Staubli VAL3: FILEDIR.pjx

--- FILEDIR.pjx ---
Parameters version=s7.7.1 stackSize=5000 millimeterUnit=true
Program file=CloseAllFile.pgx
Program file=CloseFile.pgx
Program file=CopyFileContext.pgx
Program file=CreatDir.pgx
Program file=CreatFile.pgx
Program file=Example.pgx
Program file=ExampleTest.pgx
Program file=GetLine.pgx
Program file=GetTrajFlag.pgx
Program file=ReadMe.pgx
Program file=SplitActionLine.pgx
Program file=SplitCutPreset.pgx
Program file=SplitJoint.pgx
Program file=SplitMoveC.pgx
Program file=SplitMoveJ.pgx
Program file=SplitMoveL.pgx
Program file=SplitNumS.pgx
Program file=SplitPresetLine.pgx
Program file=SplitString.pgx
Program file=SplitTrsf.pgx
Program file=start.pgx
Program file=stop.pgx
Program file=WriteLine.pgx
Data file=FileDir.dtx

--- FILEDIR.dtx ---
mdesc mNomSpeed
num nFile2ID
num nFileID
string sBuff

--- start.pgx ---
program start()
begin
  call ExampleTest()
end

--- CloseAllFile.pgx ---
public program CloseAllFile()
begin

  call CloseFile(0)
  call CloseFile(1)
  call CloseFile(2)
  call CloseFile(3)
  call CloseFile(4)
  call CloseFile(5)
  call CloseFile(6)
  call CloseFile(7)
  call CloseFile(8)
  call CloseFile(9)
  delay(0)

end

--- CloseFile.pgx ---
public program CloseFile(num x_nFileID (dimensions=1))
begin

  //文件标志符


  if x_nFileID<0 or x_nFileID>9
    return
  endIf

  //
  switch x_nFileID
    case 0
      $fileClose(0)
    break

    case 1
      $fileClose(1)
    break

    case 2
      $fileClose(2)
    break

    case 3
      $fileClose(3)
    break

    case 4
      $fileClose(4)
    break

    case 5
      $fileClose(5)
    break
    case 6
      $fileClose(6)
    break

    case 7
      $fileClose(7)
    break
    case 8
      $fileClose(8)
    break

    case 9
      $fileClose(9)
    break


  endSwitch


end

--- CopyFileContext.pgx ---
public program CopyFileContext(bool x_bRes (dimensions=1), string x_sFileSource (dimensions=1), string x_sFileDest (dimensions=1), num x_nStart (dimensions=1), num x_nEnd (dimensions=1))
  local num l_nIndex
  local num l_nNum
  local string l_sBuff
begin

  x_bRes=false
  if x_nEnd==-1
    x_nEnd=50000000
  endIf
  if x_sFileDest=="" or x_nStart<0 or x_nEnd<1 or x_nEnd<x_nStart or x_sFileDest==""
    return
  endIf
  if !$fileExists(x_sFileSource) or !$fileExists(x_sFileDest)
    return
  endIf


  nFileID=$fileOpen(x_sFileSource,"r")
  if nFileID<0 or nFileID>9
    return
  endIf

  nFile2ID=$fileOpen(x_sFileDest,"a")
  if nFile2ID<0 or nFile2ID>9
    return
  endIf


  l_nNum=1
  while true
    if $fileGet(nFileID,l_sBuff,l_nNum)!=1
      call CloseAllFile()
      return
    endIf
    if l_nIndex>=x_nStart and l_nIndex<=x_nEnd

      if $fileSet(nFile2ID,l_sBuff,l_nNum)!=1
        call CloseAllFile()
        return
      endIf
    endIf
    l_nIndex=l_nIndex+1
  endWhile

  call CloseAllFile()


end

--- CREATDIR.pgx ---
public program CreatDir(string x_sDirName (dimensions=1), bool& x_bRes (dimensions=1))
  local num l_nFileID
begin
  //说明：x_sDirName一般为 /usr/usrapp
  //
  //



  x_bRes=false
  //目录名为空则返回
  if x_sDirName==""
    return
  endIf

  //打开文件，如果文件不存在则新建文件
  l_nFileID=$fileOpen(x_sDirName+"\text","w")
  if l_nFileID<0 or l_nFileID>9
    return
  endIf
  //关闭文件
  call CloseFile(l_nFileID)
  //删除文件  保留目录
  $delete(x_sDirName+"\text")
  x_bRes=true


end

--- CreatFile.pgx ---
public program CreatFile(string x_sFileName (dimensions=1), bool& x_bRes (dimensions=1))
begin

  x_bRes=false
  nFileID=$fileOpen(x_sFileName,"w")
  if nFileID<0 or nFileID>9
    return
  endIf
  x_bRes=true
  call CloseAllFile()


end

--- EXAMPLE.pgx ---
public program Example()
  local num l_nLine
  local bool l_bBool
  local string l_sString
begin
  cls()
  title("读写文本实例")


  //*********************************************************************
  //新建文本
  gotoxy(0,0)
  put("新建文本HelloVal3.txt")
  nFileID=$fileOpen("Disk://txt/HelloVal3.txt","w")
  if nFileID<0 or nFileID>9
    gotoxy(0,1)
    put("新建打开文件出错！")
    return
  endIf

  //书写文本
  call WriteLine(nFileID,"Hello Val3!",l_bBool)
  if !l_bBool
    gotoxy(0,2)
    put("写入文件出错！")
    return
  endIf

  //关闭文件
  $fileClose(nFileID)

  //*************************************************************************
  //读取文件
  gotoxy(0,0)
  put("读取文本HelloVal3.txt")
  nFileID=$fileOpen("Disk://txt/HelloVal3.txt","r")
  if nFileID<0 or nFileID>9
    gotoxy(0,1)
    put("读取打开文件出错！")
    return
  endIf

  call GetLine(nFileID,l_sString,l_bBool)
  gotoxy(0,2)
  if !l_bBool
    put("读取文件出错！")
    return
  else
    put(l_sString)
  endIf

  //关闭文件
  $fileClose(nFileID)

  //****************************************************************************
  //添加文本
  gotoxy(0,0)
  put("添加文本HelloVal3.txt")
  nFileID=$fileOpen("Disk://txt/HelloVal3.txt","a")
  if nFileID<0 or nFileID>9
    gotoxy(0,1)
    put("添加打开文件出错！")
    return
  endIf

  //书写文本
  call WriteLine(nFileID,"Hello Val3!",l_bBool)
  if !l_bBool
    gotoxy(0,2)
    put("添加写入文件出错！")
    return
  endIf

  //关闭文件
  $fileClose(nFileID)


  //****************************************************************************
  // 删除文本
  gotoxy(0,6)
  if $delete("Disk://txt/HelloVal3.txt")
    put("删除文本成功!")
    return
  else
    put("删除文本失败!")
  endIf

end

--- ExampleTest.pgx ---
program ExampleTest()
  local num l_nStart
  local num l_nEnd
  local bool l_bRes
  local num l_nNum
  local string l_sBuff
begin


  //××××××××××××××××××××××××××××××××××××××××××××××××××××××××××××××××××××××××××××××××××××
  //××××××××××××××××××××××××××××××××××××××××××××××××××××××××××××××××××××××××××××××××××××
  //把product文件中的某条路径给替换掉
  //





  //查询
  call GetTrajFlag(l_bRes,"Disk://product1.txt",3,l_nStart,l_nEnd)
  if !l_bRes
    return
  endIf


  //产生文件
  call CreatFile("Disk://Buff.txt",l_bRes)
  if !l_bRes
    return
  endIf

  //添加开头
  call CopyFileContext(l_bRes,"Disk://product1.txt","Disk://Buff.txt",0,l_nStart-2)
  if !l_bRes
    return
  endIf
  //***************************************************************************************
  //输入内容
  nFileID=$fileOpen("Disk://Buff.txt","a")
  if nFileID<0 or nFileID>9
    return
  endIf

  l_sBuff="=BEGIN"
  l_nNum=$fileSet(nFileID,l_sBuff,l_nNum)

  for l_nNum=0 to 100
    l_sBuff=toString("",l_nNum)
    if $fileSet(nFileID,l_sBuff,1)!=1
      return
    endIf
  endFor

  l_sBuff="=END"
  l_nNum=$fileSet(nFileID,l_sBuff,l_nNum)
  call CloseAllFile()
  //************************************************************************************

  //把末尾给附加上去
  call CopyFileContext(l_bRes,"Disk://product1.txt","Disk://Buff.txt",l_nEnd+1,-1)
  if !l_bRes
    return
  endIf

  //把临时文件给删除掉
  //使用rename必须把需要命名的文件的名字不能存在，否则报错
  $delete("Disk://product1.txt")
  if !$rename("Disk://Buff.txt","Disk://product1.txt")
  endIf
end

--- GETLINE.pgx ---
public program GetLine(num x_nFileID (dimensions=1), string& x_sContext (dimensions=1), bool& x_bRes (dimensions=1))
  local num l_nNum
begin


  //文件标志符

  x_bRes=false
  if x_nFileID<0 or x_nFileID>9
    return
  endIf
  //
  switch x_nFileID
    case 0
      l_nNum=$fileGet(0,x_sContext,1)
    break

    case 1
      l_nNum=$fileGet(1,x_sContext,1)
    break

    case 2
      l_nNum=$fileGet(2,x_sContext,1)
    break

    case 3
      l_nNum=$fileGet(3,x_sContext,1)
    break

    case 4
      l_nNum=$fileGet(4,x_sContext,1)
    break

    case 5
      l_nNum=$fileGet(5,x_sContext,1)
    break
    case 6
      l_nNum=$fileGet(6,x_sContext,1)
    break

    case 7
      l_nNum=$fileGet(7,x_sContext,1)
    break
    case 8
      l_nNum=$fileGet(8,x_sContext,1)
    break

    case 9
      l_nNum=$fileGet(9,x_sContext,1)
    break


  endSwitch
  if l_nNum!=1
    return
  endIf
  x_bRes=true




end

--- GetTrajFlag.pgx ---
public program GetTrajFlag(bool& x_bRes (dimensions=1), string x_sFileName (dimensions=1), num x_nTrajIndex (dimensions=1), num& x_nStart (dimensions=1), num& x_nEnd (dimensions=1))
  local string l_sBuff
  local num l_nIndex
  local num l_nStartIndex
  local num l_nEndIndex
begin
  //参数初始化
  x_bRes=false
  x_nStart=0
  x_nEnd=0
  l_sBuff=""
  l_nIndex=0
  l_nEndIndex=0
  l_nStartIndex=0

  //传入参数合法性判断
  if x_sFileName=="" or x_nTrajIndex<1
    return
  endIf

  //打开文件
  nFileID=$fileOpen(x_sFileName,"r")
  if nFileID<0 or nFileID>9
    return
  endIf


  //查询关键字
  while !x_bRes and $fileGet(nFileID,l_sBuff,1)==1
    l_nIndex=l_nIndex+1

    if find(l_sBuff,"=BEGIN")>=0
      l_nStartIndex=l_nStartIndex+1
      x_nStart=l_nIndex
    endIf

    if find(l_sBuff,"=END")>=0
      l_nEndIndex=l_nEndIndex+1
      x_nEnd=l_nIndex
    endIf

    if l_nStartIndex==x_nTrajIndex and l_nEndIndex==x_nTrajIndex

      x_bRes=true
    endIf

  endWhile

  call CloseAllFile()

  //把所有文件给关闭掉

end

--- README.pgx ---
program ReadMe()
begin



end

--- SplitActionLine.pgx ---
public program SplitActionLine(string x_sLine, num& x_nDest[] (dimensions=3), num x_nFlag, bool& x_bRes)
  local num l_nData[25]
  local num l_nNum
  local num l_nBuff
  local string l_sChar[2]
begin

  x_bRes=false
  if x_sLine=="" or find(x_sLine,"=")<0
    return
  endIf

  x_sLine=right(x_sLine,len(x_sLine)-find(x_sLine,"=")-1)

  //如果这一行为空
  if x_sLine==""
    x_bRes=true
    return
  endIf


  //解析每一行
  l_sChar[0]=","
  l_sChar[1]=";"

  call SplitNumS(x_sLine,l_nData,l_sChar,x_bRes)

  if !x_bRes
    return
  endIf

  l_nBuff=0
  for l_nNum=0 to 11
    x_nDest[x_nFlag,l_nNum,0]=max(l_nData[l_nBuff],0)
    l_nBuff=l_nBuff+1
    x_nDest[x_nFlag,l_nNum,1]=max(l_nData[l_nBuff],0)
    l_nBuff=l_nBuff+1
  endFor





x_bRes=true






end

--- SplitCutPreset.pgx ---
public program SplitCutPreset(string x_sSLine, trsf& x_tr1, bool& x_bRes)
  local string l_sChar[2]
  local num l_nData[25]
  local num l_nIndex
begin


  x_bRes=false

  if x_sSLine==""
    return
  endIf

  x_sSLine=right(x_sSLine,len(x_sSLine)-len("MOVEL="))

  //解析每一行
  l_sChar[0]=","
  l_sChar[1]="/"
  for l_nIndex=0 to 24
    l_nData[l_nIndex]=-999999.999
  endFor

  call SplitNumS(x_sSLine,l_nData,l_sChar,x_bRes)

  if !x_bRes
    return
  endIf

  for l_nIndex=0 to 24
    if l_nData[l_nIndex]==-999999.999
      if l_nIndex<7
        return
      endIf

      x_tr1.rx=l_nData[l_nIndex-2]
      x_tr1.ry=l_nData[l_nIndex-1]
      x_bRes=true
      return


    endIf



  endFor



//  x_tr1.x=l_nData[0]
//  x_tr1.y=l_nData[1]
//  x_tr1.z=l_nData[2]
//  x_tr1.rx=l_nData[3]
//  x_tr1.ry=l_nData[4]
//  x_tr1.rz=l_nData[5]
//
//
//
//  if !x_bCut
//
//    x_trP.z=l_nData[6]
//    x_trP.rx=l_nData[7]
//  else
//    x_trP.x=l_nData[6]
//    x_trP.y=l_nData[7]
//    x_trP.z=l_nData[8]
//    x_trP.rx=l_nData[9]
//    x_trP.ry=l_nData[10]
//    //x_trP.rz=l_nData[17]
//
//  endIf




end

--- SplitJoint.pgx ---
public program SplitJoint(string x_sSLine, string x_sTitle, jointRx& x_jJ, bool& x_bRes)
  local trsf l_trTrsf
  local num l_nData[6]
  local string l_sChar[2]
begin

//  call SplitTrsf(x_sSLine,x_sTitle,l_trTrsf,x_bRes)
//  if x_bRes
//    x_jJ.j1=l_trTrsf.x
//    x_jJ.j2=l_trTrsf.y
//    x_jJ.j3=l_trTrsf.z
//    x_jJ.j4=l_trTrsf.rx
//    x_jJ.j5=l_trTrsf.ry
//    x_jJ.j6=l_trTrsf.rz
//
//  endIf


  x_bRes=false

  if x_sSLine==""
    return
  endIf

  x_sSLine=right(x_sSLine,len(x_sSLine)-len(x_sTitle))

  //解析每一行
  l_sChar[0]=","
  l_sChar[1]=","

  call SplitNumS(x_sSLine,l_nData,l_sChar,x_bRes)

  if !x_bRes
    return
  endIf

  x_jJ.j1=l_nData[0]
  x_jJ.j2=l_nData[1]
  x_jJ.j3=l_nData[2]
  x_jJ.j4=l_nData[3]
  x_jJ.j5=l_nData[4]
  x_jJ.j6=l_nData[5]






end

--- SplitMoveC.pgx ---
public program SplitMoveC(string x_sSLine (dimensions=1), trsf& x_tr1 (dimensions=1), trsf& x_tr2 (dimensions=1), trsf& x_trP (dimensions=1), bool& x_bRes (dimensions=1))
  local string l_sChar[2]
  local num l_nData[25]
begin
  x_bRes=false

  if x_sSLine==""
    return
  endIf

  x_sSLine=right(x_sSLine,len(x_sSLine)-len("MOVEC="))

  //解析每一行
  l_sChar[0]=","
  l_sChar[1]="/"

  call SplitNumS(x_sSLine,l_nData,l_sChar,x_bRes)

  if !x_bRes
    return
  endIf

  x_tr1.x=l_nData[0]
  x_tr1.y=l_nData[1]
  x_tr1.z=l_nData[2]
  x_tr1.rx=l_nData[3]
  x_tr1.ry=l_nData[4]
  x_tr1.rz=l_nData[5]

  x_tr2.x=l_nData[6]
  x_tr2.y=l_nData[7]
  x_tr2.z=l_nData[8]
  x_tr2.rx=l_nData[9]
  x_tr2.ry=l_nData[10]
  x_tr2.rz=l_nData[11]


  x_trP.x=l_nData[12]
  x_trP.y=l_nData[13]
  x_trP.z=l_nData[14]
  x_trP.rx=l_nData[15]
  x_trP.ry=l_nData[16]
  //x_trP.rz=l_nData[17]




end

--- SplitMoveJ.pgx ---
public program SplitMoveJ(string x_sSLine, joint& x_jJ, trsf& x_trP, bool x_bCut, bool& x_bRes)
  local string l_sChar[2]
  local num l_nData[25]
begin
  x_bRes=false

  if x_sSLine==""
    return
  endIf

  x_sSLine=right(x_sSLine,len(x_sSLine)-len("MOVEJ="))

  //解析每一行
  l_sChar[0]=","
  l_sChar[1]="/"

  call SplitNumS(x_sSLine,l_nData,l_sChar,x_bRes)

  if !x_bRes
    return
  endIf

  x_jJ.j1=l_nData[0]
  x_jJ.j2=l_nData[1]
  x_jJ.j3=l_nData[2]
  x_jJ.j4=l_nData[3]
  x_jJ.j5=l_nData[4]
  x_jJ.j6=l_nData[5]



  if !x_bCut

    x_trP.z=l_nData[6]
    x_trP.rx=l_nData[7]
  else
    x_trP.x=l_nData[6]
    x_trP.y=l_nData[7]
    x_trP.z=l_nData[8]
    x_trP.rx=l_nData[9]
    x_trP.ry=l_nData[10]
    //x_trP.rz=l_nData[17]

  endIf




end

--- SplitMoveL.pgx ---
public program SplitMoveL(string x_sSLine (dimensions=1), trsf& x_tr1 (dimensions=1), trsf& x_trP (dimensions=1), bool x_bCut (dimensions=1), bool& x_bRes (dimensions=1))
  local string l_sChar[2]
  local num l_nData[25]
begin
  x_bRes=false

  if x_sSLine==""
    return
  endIf

  x_sSLine=right(x_sSLine,len(x_sSLine)-len("MOVEL="))

  //解析每一行
  l_sChar[0]=","
  l_sChar[1]="/"

  call SplitNumS(x_sSLine,l_nData,l_sChar,x_bRes)

  if !x_bRes
    return
  endIf

  x_tr1.x=l_nData[0]
  x_tr1.y=l_nData[1]
  x_tr1.z=l_nData[2]
  x_tr1.rx=l_nData[3]
  x_tr1.ry=l_nData[4]
  x_tr1.rz=l_nData[5]



  if !x_bCut

    x_trP.z=l_nData[6]
    x_trP.rx=l_nData[7]
  else
    x_trP.x=l_nData[6]
    x_trP.y=l_nData[7]
    x_trP.z=l_nData[8]
    x_trP.rx=l_nData[9]
    x_trP.ry=l_nData[10]
    //x_trP.rz=l_nData[17]

  endIf




end

--- SplitNumS.pgx ---
public program SplitNumS(string x_Source (dimensions=1), num& x_Res[] (dimensions=1), string& x_sChar[] (dimensions=1), bool& x_bRes (dimensions=1))
  local num l_nNum
begin

  call SplitString(x_Source,sBuff,x_sChar,x_bRes)
  if !x_bRes
    return
  endIf



  //把分解的字符串转化为数字量
  for l_nNum=0 to min(size(sBuff)-1,size(x_Res)-1)
    toNum(sBuff[l_nNum],x_Res[l_nNum],x_bRes)
    if !x_bRes
      return
    endIf
  endFor




end

--- SplitPresetLine.pgx ---
public program SplitPresetLine(string x_sLine (dimensions=1), num& x_nDest[] (dimensions=2), num x_nFlag (dimensions=1), bool& x_bRes (dimensions=1))
  local num l_nData[25]
  local num l_nNum
  local num l_nBuff
  local string l_sChar[2]
begin

  x_bRes=false
  if x_sLine==""
    return
  endIf

  // x_sLine=right(x_sLine,len(x_sLine)-find(x_sLine,"=")-1)

  //如果这一行为空
  if x_sLine==""
    x_bRes=true
    return
  endIf


  //解析每一行
  l_sChar[0]=","
  l_sChar[1]=","

  call SplitNumS(x_sLine,l_nData,l_sChar,x_bRes)

  if !x_bRes
    return
  endIf

  l_nBuff=0
  for l_nNum=0 to 4
    //强制对工艺进行设置
    x_nDest[x_nFlag,l_nNum]=max(min(l_nData[l_nBuff],100),0)
    l_nBuff=l_nBuff+1
  endFor












end

--- SplitString.pgx ---
public program SplitString(string x_Source (dimensions=1), string& x_sDest[] (dimensions=1), string& x_sChar[] (dimensions=1), bool& x_bRes (dimensions=1))
  local num l_nResNum
  local string l_sBuff
  local num l_nFlag
  local num l_nBuff
  local num l_nIndex
begin
  //每个函数头格式
  //×××××××××××××××××××××××××××××××××××××××××××××××××
  //函数名：
  //功能：
  //参数含义:
  //使用Addon:
  //作者：
  //备注：x_sDest 只能是全局变量，因为用到了resize函数
  //日期：
  //×××××××××××××××××××××××××××××××××××××××××××××××××

  x_bRes=false
  l_nResNum=0
  resize(x_sDest,1,1)
  x_sDest=""
  if x_Source=="" or x_sChar==""
    return
  endIf

  l_sBuff=x_Source
  while true
    l_nFlag=10000
    //获得最小标志符序号
    for l_nIndex=0 to size(x_sChar)-1 step 1
      l_nBuff=find(l_sBuff,x_sChar[l_nIndex])
      if l_nBuff>=0 and l_nBuff<l_nFlag
        l_nFlag=l_nBuff
      endIf
    endFor


    //里面没有标志符
    if len(l_sBuff)>=1 and l_nFlag==10000
      if l_nResNum!=0
        resize(x_sDest,1,l_nResNum+1)
      endIf
      x_sDest[l_nResNum]=l_sBuff
      x_bRes=true
      return
    endIf

    //字符串为空
    if l_sBuff==""
      x_bRes=true
      return
    endIf


    //分开
    if l_nFlag==0
      l_sBuff=right(l_sBuff,len(l_sBuff)-1)
    else
      if l_nResNum!=0
        resize(x_sDest,1,l_nResNum+1)
      endIf
      x_sDest[l_nResNum]=left(l_sBuff,l_nFlag)
      l_nResNum=l_nResNum+1
      l_sBuff=right(l_sBuff,len(l_sBuff)-l_nFlag-1)
    endIf
  endWhile


end

--- SplitTrsf.pgx ---
public program SplitTrsf(string x_sSLine (dimensions=1), string x_sTitle (dimensions=1), trsf& x_trTrsf (dimensions=1), bool& x_bRes (dimensions=1))
  local string l_sChar[2]
  local num l_nData[25]
begin
  x_bRes=false

  if x_sSLine==""
    return
  endIf

  x_sSLine=right(x_sSLine,len(x_sSLine)-len(x_sTitle))

  //解析每一行
  l_sChar[0]=","
  l_sChar[1]=","

  call SplitNumS(x_sSLine,l_nData,l_sChar,x_bRes)

  if !x_bRes
    return
  endIf

  x_trTrsf.x=l_nData[0]
  x_trTrsf.y=l_nData[1]
  x_trTrsf.z=l_nData[2]
  x_trTrsf.rx=l_nData[3]
  x_trTrsf.ry=l_nData[4]
  x_trTrsf.rz=l_nData[5]




end

--- WriteLine.pgx ---
public program WriteLine(num x_nFileID (dimensions=1), string x_sContext (dimensions=1), bool& x_bRes (dimensions=1))
  local num l_nNum
  local string l_sString
begin

  //文件标志符

  x_bRes=false
  if x_nFileID<0 or x_nFileID>9
    return
  endIf
  l_sString[0]=x_sContext
  //
  switch x_nFileID
    case 0
      l_nNum=$fileSet(0,l_sString,1)
    break

    case 1
      l_nNum=$fileSet(1,l_sString,1)
    break

    case 2
      l_nNum=$fileSet(2,l_sString,1)
    break

    case 3
      l_nNum=$fileSet(3,l_sString,1)
    break

    case 4
      l_nNum=$fileSet(4,l_sString,1)
    break

    case 5
      l_nNum=$fileSet(5,l_sString,1)
    break
    case 6
      l_nNum=$fileSet(6,l_sString,1)
    break

    case 7
      l_nNum=$fileSet(7,l_sString,1)
    break
    case 8
      l_nNum=$fileSet(8,l_sString,1)
    break

    case 9
      l_nNum=$fileSet(9,l_sString,1)
    break


  endSwitch
  if l_nNum!=1
    return
  endIf
  x_bRes=true


end
